(* CODESYS project ATV32_EIP_LMCx00C_V003.project
   Company: Schneider Electric
   DefaultNamespace: QuickMotionProgramming
   Title: QuickMotionProgramming
   Description: Demoproject for QuickMotionProgramming
   Author: Schneider Electric Automation GmbH
   Version: 1.0.6.0

Project tree, tasks and I/O mapping:
  LMC_PacDrive : PacDrive LMC 300/400/600C, Schneider Electric, order no. LMCx00C, version 1.51.10.0
    application Application
      libraries: PD_GlobalDiagnostics, 1.2.0.0 (Schneider Electric); PD_PacDriveLib, 1.4.9.0 (Schneider Electric); PD_AxisModule, 1.3.5.0 (Schneider Electric); PD_Template, 1.3.3.0 (Schneider Electric)
      task TASK_SR_MainMachine (cyclic, interval T#10ms, priority 8, watchdog T#100ms x 10) calls SR_MainMachine
      GlobalVariables/
        global variables RestoreAxisPosition
        global variables GlobalVariables_Machine
        global variables Global_ATV32
        global variables Logging
        global variables HardwareInOuts
        global variables InputVariablesSLB
        global variables InputVariablesExt
        global variables ExceptionHandling
        global variables Diagnostics
      ProjectDiagnostics/
        function FC_EtDiagExtUserToString [ST]
        data type ET_DiagExtUser
        data type ET_DiagExt
        function FC_EtDiagExtToString [ST]
      000 Program/
        00 Task Calls/
          program SR_MainMachine [LD]: Logic_ATV32
      Data Types/
        data type ET_Cmd
        data type ET_ATV32CmdWord
        data type ET_ATV32StatusWord
      300 EIP Utilities/
        function FC_EIPWriteWORDtoBYTES [ST]
        function FC_EIPReadWORDfromBYTES [ST]
    EPAS Mechatronic
    EPAS SERCOSIII Device Commissioning
    Message Logger
    SERCOSIII : SERCOS III Interface, Schneider Electric, version 1.51.10.0
      DRV_Master : Lexium LXM62 Drive, Schneider Electric, order no. LXM62DU60, LXM62DD15, LXM62DD27, LXM62DD45, LXM62DC13, version 1.51.10.0
          settings: ConfiguredPowerSupply = 'PSM_Lexium62'
      DRV_Axis1 : Lexium LXM62 Drive, Schneider Electric, order no. LXM62DU60, LXM62DD15, LXM62DD27, LXM62DD45, LXM62DC13, version 1.51.10.0
          settings: ConfiguredPowerSupply = 'PSM_Lexium62'
      DRV_Axis2 : Lexium LXM62 Drive, Schneider Electric, order no. LXM62DU60, LXM62DD15, LXM62DD27, LXM62DD45, LXM62DC13, version 1.51.10.0
          settings: ConfiguredPowerSupply = 'PSM_Lexium62'
      PSM_Lexium62 : Lexium LXM62 Power Supply, Schneider Electric, order no. LXM62PD84, LXM62PD20, version 1.51.10.0
    DIG_DigitalIn : Digital Inputs, Schneider Electric, version 1.51.10.0
      DI_11 : Input, Schneider Electric, version 1.51.10.0
      DI_2 : Input, Schneider Electric, version 1.51.10.0
      DI_10 : Input, Schneider Electric, version 1.51.10.0
      DI_19 : Input, Schneider Electric, version 1.51.10.0
      DI_5 : Input, Schneider Electric, version 1.51.10.0
      DI_17 : Input, Schneider Electric, version 1.51.10.0
      DI_0 : Input, Schneider Electric, version 1.51.10.0
      DI_8 : Input, Schneider Electric, version 1.51.10.0
      DI_1 : Input, Schneider Electric, version 1.51.10.0
      ADI_0 : Fast Input, Schneider Electric, version 1.51.10.0
      ADI_1 : Fast Input, Schneider Electric, version 1.51.10.0
      DI_9 : Input, Schneider Electric, version 1.51.10.0
      DI_12 : Input, Schneider Electric, version 1.51.10.0
      DI_15 : Input, Schneider Electric, version 1.51.10.0
      DI_6 : Input, Schneider Electric, version 1.51.10.0
      DI_13 : Input, Schneider Electric, version 1.51.10.0
      DI_14 : Input, Schneider Electric, version 1.51.10.0
      ADI_2 : Fast Input, Schneider Electric, version 1.51.10.0
      ADI_3 : Fast Input, Schneider Electric, version 1.51.10.0
      DI_7 : Input, Schneider Electric, version 1.51.10.0
      DI_4 : Input, Schneider Electric, version 1.51.10.0
      DI_16 : Input, Schneider Electric, version 1.51.10.0
      DI_18 : Input, Schneider Electric, version 1.51.10.0
      DI_3 : Input, Schneider Electric, version 1.51.10.0
    DQG_DigitalOut : Digital Outputs, Schneider Electric, version 1.51.10.0
        settings: DiagMask = 2#1111111100000000; OpenloadDiagMsk = 2#1111111100000000
      DQ_1 : Output, Schneider Electric, version 1.51.10.0
      DQ_0 : Output, Schneider Electric, version 1.51.10.0
      DQ_6 : Output, Schneider Electric, version 1.51.10.0
      DQ_4 : Output, Schneider Electric, version 1.51.10.0
      DQ_9 : Output, Schneider Electric, version 1.51.10.0
      DQ_13 : Output, Schneider Electric, version 1.51.10.0
      DQ_14 : Output, Schneider Electric, version 1.51.10.0
      DQ_15 : Output, Schneider Electric, version 1.51.10.0
      DQ_10 : Output, Schneider Electric, version 1.51.10.0
      DQ_5 : Output, Schneider Electric, version 1.51.10.0
      DQ_12 : Output, Schneider Electric, version 1.51.10.0
      DQ_11 : Output, Schneider Electric, version 1.51.10.0
      DQ_2 : Output, Schneider Electric, version 1.51.10.0
      DQ_3 : Output, Schneider Electric, version 1.51.10.0
      DQ_8 : Output, Schneider Electric, version 1.51.10.0
      DQ_7 : Output, Schneider Electric, version 1.51.10.0
    AI_0 : Analog Input, Schneider Electric, version 1.51.10.0
    AI_1 : Analog Input, Schneider Electric, version 1.51.10.0
    AQ_1 : Analog Output, Schneider Electric, version 1.51.10.0
    TPG_TPIn : Touch Probe Inputs, Schneider Electric, version 1.51.10.0
      TP_3 : Touch Probe Input, Schneider Electric, version 1.51.10.0
      TP_9 : Touch Probe Input, Schneider Electric, version 1.51.10.0
      TP_4 : Touch Probe Input, Schneider Electric, version 1.51.10.0
      TP_5 : Touch Probe Input, Schneider Electric, version 1.51.10.0
      TP_6 : Touch Probe Input, Schneider Electric, version 1.51.10.0
      TP_14 : Touch Probe Input, Schneider Electric, version 1.51.10.0
      TP_7 : Touch Probe Input, Schneider Electric, version 1.51.10.0
      TP_15 : Touch Probe Input, Schneider Electric, version 1.51.10.0
      TP_8 : Touch Probe Input, Schneider Electric, version 1.51.10.0
      TP_12 : Touch Probe Input, Schneider Electric, version 1.51.10.0
      TP_13 : Touch Probe Input, Schneider Electric, version 1.51.10.0
      TP_11 : Touch Probe Input, Schneider Electric, version 1.51.10.0
      TP_0 : Touch Probe Input, Schneider Electric, version 1.51.10.0
      TP_1 : Touch Probe Input, Schneider Electric, version 1.51.10.0
      TP_2 : Touch Probe Input, Schneider Electric, version 1.51.10.0
      TP_10 : Touch Probe Input, Schneider Electric, version 1.51.10.0
    AQ_0 : Analog Output, Schneider Electric, version 1.51.10.0
    LE_Master : Log. Encoder, Schneider Electric, version 1.51.10.0
    LE_Axis1 : Log. Encoder, Schneider Electric, version 1.51.10.0
    LE_Axis2 : Log. Encoder, Schneider Electric, version 1.51.10.0
    EIPS_Scanner : EtherNet-IP-Scanner, Schneider Electric, version 1.51.10.0
        settings: IPAddress = [16#C0,16#A8,16#01,16#0A]; SubnetMask = [16#FF,16#FF,16#FF,16#00]; GatewayAddress = [16#00,16#00,16#00,16#00]
      ATV32 : ATV32, Schneider Electric, version Major Revision=16#1, Minor Revision = 16#7
          settings: INITIALIZED = TRUE; IP address of Target = [16#C0,16#A8,16#01,16#14]; MAC address of Target = [16#00,16#00,16#00,16#00,16#00,16#00]; Keying.Check Minor Revision = FALSE; Number of Connections = 1; Connection Settings.Requested packet intervall (µs) = 10000; Connection Settings.OT Connection Parameters = 18450; Connection Settings.TO Connection Parameters = 10254; Connection Settings.Connection Flags = 1056; Connection Settings.Connection Path Size = 8; Connection Path = [16#20,16#04,16#24,16#05,16#2C,16#64,16#2C,16#65]
          input  Application.g_abATV32_1_StatusWordBytes[1] : BYTE  // Input0
          input  Application.g_abATV32_1_StatusWordBytes[2] : BYTE  // Input1
          input  Application.g_abATV32_1_ActVelocityBytes[1] : BYTE  // Input2
          input  Application.g_abATV32_1_ActVelocityBytes[2] : BYTE  // Input3
          output Application.g_abATV32_1_CommandWordBytes[1] : BYTE  // Output0
          output Application.g_abATV32_1_CommandWordBytes[2] : BYTE  // Output1
          output Application.g_abATV32_1_CmdVelocityBytes[1] : BYTE  // Output2
          output Application.g_abATV32_1_CmdVelocityBytes[2] : BYTE  // Output3
          unmapped channels: Input4, Input5, Input6, Input7, Input8, Input9, Input10, Input11, Output4, Output5, Output6, Output7, Output8, Output9, Output10, Output11
  Project Information/
    function GetVersion [ST]
    function GetBooleanProperty [ST]
    function GetTitle [ST]
    function GetVersionProperty [ST]
    function GetTextProperty [ST]
    function GetCompany [ST]
    function GetNumberProperty [ST]
  MainMachine
    DRV_Master
      Drive
    DRV_Axis2
      Drive
    DRV_Axis1
      Drive
    PSM_Lexium62
  MainMachine
    DRV_Master
      Drive
    DRV_Axis1
      Drive
    DRV_Axis2
      Drive
    PSM_Lexium62
  text list GlobalTextList
*)

// LMC_PacDrive/Application/ProjectDiagnostics/ET_DiagExtUser
{attribute 'qualified_only'}
TYPE ET_DiagExtUser :
(
(* Minimum value +0 *)
	Exception1FromEquipmentModule		:= 0,
	Exception2FromEquipmentModule		:= 1,
	
	Exception1FromMain					:= 2,
	Exception2FromMain					:= 3,
	Exception3FromMain					:= 4,
	Exception4FromMain					:= 5,
	Exception5FromMain					:= 6
)UDINT;
END_TYPE

// LMC_PacDrive/Application/ProjectDiagnostics/ET_DiagExt
{attribute 'qualified_only'}
TYPE ET_DiagExt :
(  
	(* Minimum value +0 *)
	Ok								:= 0,
	Disabled						:= 1,
	WaitUntilControllerFinishedBoot	:= 2,
	Initializing					:= 3,
	DeactivatingSubModules			:= 4,
	ExecuteStep						:= 5,
	WaitAtNegativeStep				:= 6,
	WaitCmdsDone					:= 7,
	WaitForCmd						:= 8,
	SubModuleInException			:= 9,
	ModuleControllerException		:= 10,
	UnknownStateModuleController	:= 11,
	
	SystemFatalException			:= 12,
	SystemException					:= 13,
	SystemWarning					:= 14,
	MainSystemEmergencyStop			:= 15,
	InvalidPointer					:= 16,	
	UpdateStructsException			:= 17,
	InitReactionsException			:= 18,
	InitSubModulesException			:= 19,
	DriveInvalid					:= 20,
	UnknownDiagExt					:= 21,
	
	Exception1FromVis				:= 22,
	Exception2FromVis				:= 23,
	Exception3FromVis				:= 24,
	Exception4FromVis				:= 25,
	Exception5FromVis				:= 26,
	
	DiagnosticsWarning					:= 27,
	WaitUntilDiagnosticsManagerReady	:= 28,
	WaitUntilDisabled					:= 29,
	WaitUntilDiagSourceRegistered		:= 30,
	WaitForCommunication				:= 31,
	DataSuccessfullyWritten				:= 32,
	WritingToFile						:= 33,
	FileIdInvalid						:= 34,
	CmdUnknown							:= 35,	
	UnexpectedFeedback					:= 36,
	UnknownDiagExtUser					:= 37,
	
	ExceptionListOverflow				:= 50
	
)UDINT;
END_TYPE

// LMC_PacDrive/Application/Data Types/ET_Cmd
{attribute 'qualified_only'}
TYPE ET_Cmd :
(	NoCmd				:= 0,

	(* TPL.Gc_udiUserCmdOffset : UDINT := 25000; // >= 25000: user defined Commands *)
	DriveEnableOn		:= 25999,
	DriveEnableOff		:= 25998,
	Init				:= 25997,
	Prepare				:= 25996,
	Production			:= 25995,
	Auto				:= 25994,
	BrakeRelease		:= 25993,
	Abort				:= 25992,
	Standby				:= 25991,
	Manual				:= 25990,
	Jogging				:= 25989,
	Hold				:= 25988,
	Stop				:= 25987,
	Start				:= 25986,
	HoldJM				:= 25985
);
END_TYPE

// LMC_PacDrive/Application/Data Types/ET_ATV32CmdWord
TYPE ET_ATV32CmdWord :
(
	Bit0_SwitchOn := 0,
	Bit1_EnableVoltage := 1,
	Bit2_QuickStop := 2,
	Bit3_EnableOperation := 3,
	Bit4_CmdUnused,
	Bit5_CmdUnused,
	Bit6_CmdUnused,
	Bit7_FaultReset,
	Bit8_Halt,
	Bit9_CmdUnused,
	Bit10_CmdUnused,
	Bit11_FwdRev,
	Bit12_CmdUnused,
	Bit13_CmdUnused,
	Bit14_CmdUnused,
	Bit15_CmdUnused
	
);
END_TYPE

// LMC_PacDrive/Application/Data Types/ET_ATV32StatusWord
TYPE ET_ATV32StatusWord :
(
	Bit0_ReadyToSwitchOn := 0,
	Bit1_SwitchedOn := 1,
	Bit2_OperationEnabled := 2,
	Bit3_Fault := 3,
	Bit4_VoltageEnabled,
	Bit5_QuickStop,
	Bit6_SwitchOnDisabled,
	Bit7_Warning,
	Bit8_StsUnused,
	Bit9_CmdViaNetwork,
	Bit10_TargetReached,
	Bit11_LimitActive,
	Bit12_StsUnused,
	Bit13_StsUnused,
	Bit14_StsUnused,
	Bit15_StsUnused
	
);
END_TYPE

// LMC_PacDrive/Application/GlobalVariables/RestoreAxisPosition
VAR_GLOBAL PERSISTENT RETAIN
	Grp_stRestorePositionMaster	: PDL.ST_AxisRestorePosition;
	Grp_stRestorePositionAxis1	: PDL.ST_AxisRestorePosition;
	Grp_stRestorePositionAxis2	: PDL.ST_AxisRestorePosition;
	Grp_stRestorePositionAxis3	: PDL.ST_AxisRestorePosition;
	Grp_stRestorePositionMaster2: PDL.ST_AxisRestorePosition;
	Grp_stRestorePositionAxis4	: PDL.ST_AxisRestorePosition;
	Grp_stRestorePositionAxis5	: PDL.ST_AxisRestorePosition;
	Grp_stRestorePositionAxis6	: PDL.ST_AxisRestorePosition;	
END_VAR

// LMC_PacDrive/Application/GlobalVariables/GlobalVariables_Machine
VAR_GLOBAL
	g_xAllServosHomeOk			:BOOL;
END_VAR

// LMC_PacDrive/Application/GlobalVariables/Global_ATV32
VAR_GLOBAL
	g_wATV32_1_CommandVelocity:		WORD;
	g_wATV32_1_ActVelocity:		WORD;

	g_abATV32_1_CommandWordBytes:	ARRAY[1..2] OF BYTE;
	g_axATV32_1CommandWord:			ARRAY[0..15] OF BOOL;
	g_wATV32_1_CommandWord:			WORD;

	g_abATV32_1_StatusWordBytes:	ARRAY[1..2] OF BYTE;
	g_axATV32_1StatusWord:			ARRAY[0..15] OF BOOL;
	g_wATV32_1_StatusWord:			WORD;
	
	g_abATV32_1_CmdVelocityBytes:	ARRAY[1..2] OF BYTE;
	g_abATV32_1_ActVelocityBytes:	ARRAY[1..2] OF BYTE;	
END_VAR

// LMC_PacDrive/Application/GlobalVariables/Logging
VAR_GLOBAL
	G_stLogDataList			: TPL.ST_LogDataList;			(* Global log data list *)
	G_stLogDataListAscii	: TPL.ST_LogDataListAscii;		(* Temp.list for save in XML format *)
	G_stLoggerInterface		: TPL.ST_LoggerInterface;		(* Interface between logger and main machine *)
END_VAR

// LMC_PacDrive/Application/GlobalVariables/HardwareInOuts
VAR_GLOBAL
	G_xMainsContactorOut 		(*-AT %QX0.0-*)	: BOOL;

	G_xEmergencyIn  			(*-AT %IX0.0-*)	: BOOL;
	G_xMainsContactorIn 		(*-AT %IX0.1-*)	: BOOL;
END_VAR

// LMC_PacDrive/Application/GlobalVariables/InputVariablesSLB
VAR_GLOBAL
	(* SoMachine Motion Logic Builder (SLB) input *)
	G_xStartSlb				 	: BOOL;
	G_xStopSlb					: BOOL;
	G_xPrepareSlb				: BOOL;
	G_xAutoSlb					: BOOL;
	G_xHoldSlb					: BOOL;
	G_xAbortSlb					: BOOL;
	G_xProductsOkSlb			: BOOL;
	G_xPowerOnSlb				: BOOL;
	G_xPowerOffSlb				: BOOL;
	G_xManualSlb				: BOOL;
	G_xJogMachineSlb			: BOOL;
	G_xDiagQuitSlb				: BOOL;
	G_xEmergencySlb				: BOOL := TRUE;
	G_xJogForwSlb				: BOOL;
	G_xJogBackSlb				: BOOL;
	G_xBrakeReleaseSlb			: BOOL;
	
	G_udiManualModuleSelect		: UDINT;

	G_xDoEnableVis				: BOOL;

	G_xDoPrepare 				: BOOL;
	G_xDoAuto	 				: BOOL;
	G_xDoManual 				: BOOL;
	G_xDoJogMachine 			: BOOL;
	G_xDoBrakeRelease			: BOOL;

	G_xPrepareActive 			: BOOL;
	G_xAutoActive	 			: BOOL;
	G_xManualActive 			: BOOL;
	G_xJogMachineActive 		: BOOL;
	G_xBrakeReleaseActive		: BOOL;
END_VAR

// LMC_PacDrive/Application/GlobalVariables/InputVariablesExt
VAR_GLOBAL
	(* Extern / HMI input *)
	G_xStartExt			: BOOL;
	G_xStopExt			: BOOL;
	G_xPrepareExt		: BOOL;
	G_xAutoExt			: BOOL;
	G_xHoldExt			: BOOL;
	G_xAbortExt			: BOOL;
	G_xProductsOkExt	: BOOL;
	G_xPowerOnExt		: BOOL;
	G_xPowerOffExt		: BOOL;
	G_xManualExt		: BOOL;
	G_xJogMachineExt	: BOOL;
	G_xDiagQuitExt		: BOOL;
	G_xJogForwExt		: BOOL;
	G_xJogBackExt		: BOOL;
	G_xBrakeReleaseExt	: BOOL;
END_VAR

// LMC_PacDrive/Application/GlobalVariables/ExceptionHandling
VAR_GLOBAL
	G_stExceptionList		: TPL.ST_ExceptionList;
END_VAR

// LMC_PacDrive/Application/GlobalVariables/Diagnostics
VAR_GLOBAL
	G_stDiagnosticsToApplicationMarkerarea AT %MB0 : TPL.ST_DiagnosticsToApplicationMarkerArea;
END_VAR

// LMC_PacDrive/Application/000 Program/00 Task Calls/SR_MainMachine
PROGRAM SR_MainMachine
VAR
END_VAR

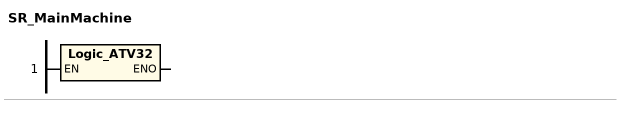
// NETWORK 1
Logic_ATV32();

ACTION Logic_ATV32:




g_wATV32_1_CommandWord := PDL.FC_PackWord(
											i_xB15:= g_axATV32_1CommandWord[Bit15_CmdUnused], 
											i_xB14:= g_axATV32_1CommandWord[Bit14_CmdUnused], 
											i_xB13:= g_axATV32_1CommandWord[Bit13_CmdUnused], 
											i_xB12:= g_axATV32_1CommandWord[Bit12_CmdUnused], 
											i_xB11:= g_axATV32_1CommandWord[Bit11_FwdRev], 
											i_xB10:= g_axATV32_1CommandWord[Bit10_CmdUnused], 
											i_xB09:= g_axATV32_1CommandWord[Bit9_CmdUnused], 
											i_xB08:= g_axATV32_1CommandWord[Bit8_Halt], 
											i_xB07:= g_axATV32_1CommandWord[Bit7_FaultReset], 
											i_xB06:= g_axATV32_1CommandWord[Bit6_CmdUnused], 
											i_xB05:= g_axATV32_1CommandWord[Bit5_CmdUnused], 
											i_xB04:= g_axATV32_1CommandWord[Bit4_CmdUnused], 
											i_xB03:= g_axATV32_1CommandWord[Bit3_EnableOperation], 
											i_xB02:= g_axATV32_1CommandWord[Bit2_QuickStop], 
											i_xB01:= g_axATV32_1CommandWord[Bit1_EnableVoltage], 
											i_xB00:= g_axATV32_1CommandWord[Bit0_SwitchOn]);

								
// Write the Command Word - FC_EIPWriteWORDtoBYTES allows us to send a word vlaue to two consecutive bytes in memory
FC_EIPWriteWORDtoBYTES(pdiSourceWord:= ADR(g_wATV32_1_CommandWord), pDestByte:=ADR(g_abATV32_1_CommandWordBytes[1]) );											

// Write the Command Velocity - FC_EIPWriteWORDtoBYTES allows us to send a word vlaue to two consecutive bytes in memory
FC_EIPWriteWORDtoBYTES(pdiSourceWord:= ADR(g_wATV32_1_CommandVelocity), pDestByte:=ADR(g_abATV32_1_CmdVelocityBytes[1]) );

// Read The Status Word - FC_EIPReadWORDFromBYTES allows us to read a word vlaue to two consecutive bytes in memory
g_wATV32_1_StatusWord := FC_EIPReadWORDfromBYTES(pByteSource:=ADR(g_abATV32_1_StatusWordBytes[1]));
	
PDL.FC_UnpackWord(i_wInput:= g_wATV32_1_StatusWord, 
				  	q_xB15=> g_axATV32_1StatusWord[Bit15_StsUnused], 
				  	q_xB14=> g_axATV32_1StatusWord[Bit14_StsUnused], 
					q_xB13=> g_axATV32_1StatusWord[Bit13_StsUnused], 
					q_xB12=> g_axATV32_1StatusWord[Bit12_StsUnused], 
					q_xB11=> g_axATV32_1StatusWord[Bit11_LimitActive], 
					q_xB10=> g_axATV32_1StatusWord[Bit10_TargetReached], 
					q_xB09=> g_axATV32_1StatusWord[Bit9_CmdViaNetwork], 
					q_xB08=> g_axATV32_1StatusWord[Bit8_StsUnused], 
					q_xB07=> g_axATV32_1StatusWord[Bit7_Warning], 
					q_xB06=> g_axATV32_1StatusWord[Bit6_SwitchOnDisabled], 
					q_xB05=> g_axATV32_1StatusWord[Bit5_QuickStop], 
					q_xB04=> g_axATV32_1StatusWord[Bit4_VoltageEnabled], 
					q_xB03=> g_axATV32_1StatusWord[Bit3_Fault], 
					q_xB02=> g_axATV32_1StatusWord[Bit2_OperationEnabled], 
					q_xB01=> g_axATV32_1StatusWord[Bit1_SwitchedOn], 
					q_xB00=> g_axATV32_1StatusWord[Bit0_ReadyToSwitchOn]);
					
// Read Actual Velocity - FC_EIPReadWORDFromBYTES allows us to read a word vlaue to two consecutive bytes in memory					
					
g_wATV32_1_ActVelocity := FC_EIPReadWORDfromBYTES(pByteSource:=ADR(g_abATV32_1_ActVelocityBytes[1]));
END_ACTION

END_PROGRAM

// LMC_PacDrive/Application/300 EIP Utilities/FC_EIPWriteWORDtoBYTES
FUNCTION FC_EIPWriteWORDtoBYTES : WORD
(* This function will write to a WORD to 2 succesive Bytes starting from the input var "pdiDestByte"
	When calling the function, "pDestByte" should be the address of an index from an ARRAY OF BYTE, then the function
	will build the WORD based on the data from the index you start with plus the next indexes in order from the array.

	Example:

	Declaration:    MyByteArray:			ARRAY[1..128] OF BYTE;

	Function Call:        FC_EIPWriteWORDtoBYTES(pdiSourceWord:= ADR(MyWORDVariable), pDestByte:= ADR(MyByteArray[1]));
*)
VAR_INPUT
	pdiSourceWord:		POINTER TO WORD;
	pDestByte:			POINTER TO WORD;
END_VAR
VAR
END_VAR

pDestByte^ := pdiSourceWord^;

END_FUNCTION

// LMC_PacDrive/Application/300 EIP Utilities/FC_EIPReadWORDfromBYTES
FUNCTION FC_EIPReadWORDfromBYTES : WORD
(* 

	Exp:
	Declaration:    MyByteArray:			ARRAY[1..128] OF BYTE;

	Function Call:        OutputDINTVaraible := FC_EIPReadWORDfromBYTES(ADR(MyByteArray[1]);
*)
VAR_INPUT
	pByteSource:		POINTER TO WORD;
END_VAR
VAR
END_VAR

FC_EIPReadWORDfromBYTES := pByteSource^;

END_FUNCTION

// Project Information/GetVersion
// This function has been automatically generated from the project information.
{attribute 'signature_flag' := '1073741824'}
{attribute 'register_in_runtime'}
FUNCTION GetVersion : VERSION
VAR_INPUT
	
END_VAR

GetVersion.uiMajor := 1;
GetVersion.uiMinor := 0;
GetVersion.uiServicePack := 6;
GetVersion.uiPatch := 0;

END_FUNCTION

// Project Information/GetBooleanProperty
// This function has been automatically generated from the project information.
{attribute 'signature_flag' := '1073741824'}
{attribute 'register_in_runtime'}
FUNCTION GetBooleanProperty : BOOL
VAR_INPUT
	stKey: WSTRING;
END_VAR

GetBooleanProperty := FALSE;

END_FUNCTION

// Project Information/GetTitle
// This function has been automatically generated from the project information.
{attribute 'signature_flag' := '1073741824'}
{attribute 'register_in_runtime'}
FUNCTION GetTitle : WSTRING
VAR_INPUT
	
END_VAR

GetTitle := "QuickMotionProgramming";

END_FUNCTION

// Project Information/GetVersionProperty
// This function has been automatically generated from the project information.
{attribute 'signature_flag' := '1073741824'}
{attribute 'register_in_runtime'}
FUNCTION GetVersionProperty : VERSION
VAR_INPUT
	stKey: WSTRING;
END_VAR

IF stKey = "Version" THEN
	GetVersionProperty.uiMajor := 1;
	GetVersionProperty.uiMinor := 0;
	GetVersionProperty.uiServicePack := 6;
	GetVersionProperty.uiPatch := 0;
ELSE
	GetVersionProperty.uiMajor := 0;
	GetVersionProperty.uiMinor := 0;
	GetVersionProperty.uiServicePack := 0;
	GetVersionProperty.uiPatch := 0;
END_IF

END_FUNCTION

// Project Information/GetTextProperty
// This function has been automatically generated from the project information.
{attribute 'signature_flag' := '1073741824'}
{attribute 'register_in_runtime'}
FUNCTION GetTextProperty : WSTRING
VAR_INPUT
	stKey: WSTRING;
END_VAR

IF stKey = "Author" THEN
	GetTextProperty := "Schneider Electric Automation GmbH";
ELSIF stKey = "Company" THEN
	GetTextProperty := "Schneider Electric";
ELSIF stKey = "DefaultNamespace" THEN
	GetTextProperty := "QuickMotionProgramming";
ELSIF stKey = "Description" THEN
	GetTextProperty := "Demoproject for QuickMotionProgramming";
ELSIF stKey = "Project" THEN
	GetTextProperty := "ATV32_EIP_LMCx00C_V003";
ELSIF stKey = "Title" THEN
	GetTextProperty := "QuickMotionProgramming";
ELSE
	GetTextProperty := "";
END_IF

END_FUNCTION

// Project Information/GetCompany
// This function has been automatically generated from the project information.
{attribute 'signature_flag' := '1073741824'}
{attribute 'register_in_runtime'}
FUNCTION GetCompany : WSTRING
VAR_INPUT
	
END_VAR

GetCompany := "Schneider Electric";

END_FUNCTION

// Project Information/GetNumberProperty
// This function has been automatically generated from the project information.
{attribute 'signature_flag' := '1073741824'}
{attribute 'register_in_runtime'}
FUNCTION GetNumberProperty : DINT
VAR_INPUT
	stKey: WSTRING;
END_VAR

GetNumberProperty := 0;

END_FUNCTION

// LMC_PacDrive/Application/ProjectDiagnostics/FC_EtDiagExtUserToString
FUNCTION FC_EtDiagExtUserToString : STRING[80]

VAR_INPUT
	i_etDiagExt : ET_DiagExtUser;
END_VAR

VAR_OUTPUT
	q_etDiag	: GD.ET_Diag := GD.ET_Diag.Ok;
	q_etDiagExt	: ET_DiagExt := ET_DiagExt.Ok;
END_VAR

VAR
END_VAR

CASE i_etDiagExt OF
	ET_DiagExtUser.Exception1FromEquipmentModule	: FC_EtDiagExtUserToString := 'Exception1FromEquipmentModule';
	ET_DiagExtUser.Exception2FromEquipmentModule	: FC_EtDiagExtUserToString := 'Exception2FromEquipmentModule';
	
	ET_DiagExtUser.Exception1FromMain				: FC_EtDiagExtUserToString := 'Exception1FromMain';
	ET_DiagExtUser.Exception2FromMain				: FC_EtDiagExtUserToString := 'Exception2FromMain';
	ET_DiagExtUser.Exception3FromMain				: FC_EtDiagExtUserToString := 'Exception3FromMain';
	ET_DiagExtUser.Exception4FromMain				: FC_EtDiagExtUserToString := 'Exception4FromMain';
	ET_DiagExtUser.Exception5FromMain				: FC_EtDiagExtUserToString := 'Exception5FromMain';
ELSE
	FC_EtDiagExtUserToString := CONCAT('Unkown ET_DiagExtUser ', UDINT_TO_STRING(i_etDiagExt));
		
	q_etDiag	:= GD.ET_Diag.InputParameterInvalid;
	q_etDiagExt	:= ET_DiagExt.UnknownDiagExtUser;
END_CASE

END_FUNCTION

// LMC_PacDrive/Application/ProjectDiagnostics/FC_EtDiagExtToString
FUNCTION FC_EtDiagExtToString : STRING[80]

VAR_INPUT
	i_etDiagExt : ET_DiagExt;
END_VAR

VAR_OUTPUT
	q_etDiag	: GD.ET_Diag := GD.ET_Diag.Ok;
	q_etDiagExt	: ET_DiagExt := ET_DiagExt.Ok;
END_VAR

VAR
END_VAR

CASE i_etDiagExt OF
	ET_DiagExt.Ok:								FC_EtDiagExtToString := 'Ok';
	ET_DiagExt.Disabled:						FC_EtDiagExtToString := 'Disabled';
	ET_DiagExt.WaitUntilControllerFinishedBoot:	FC_EtDiagExtToString := 'WaitUntilControllerFinishedBoot';
	ET_DiagExt.Initializing:					FC_EtDiagExtToString := 'Initializing';
	ET_DiagExt.DeactivatingSubModules:			FC_EtDiagExtToString := 'DeactivatingSubModules';
	ET_DiagExt.ExecuteStep:						FC_EtDiagExtToString := 'ExecuteStep';
	ET_DiagExt.WaitAtNegativeStep:				FC_EtDiagExtToString := 'WaitAtNegativeStep';
	ET_DiagExt.WaitCmdsDone:					FC_EtDiagExtToString := 'WaitCmdsDone';
	ET_DiagExt.WaitForCmd:						FC_EtDiagExtToString := 'WaitForCmd';
	ET_DiagExt.SubModuleInException:			FC_EtDiagExtToString := 'SubModuleInException';
	ET_DiagExt.ModuleControllerException:		FC_EtDiagExtToString := 'ModuleControllerException';
	ET_DiagExt.UnknownStateModuleController:	FC_EtDiagExtToString := 'UnknownStateModuleController';
	
	ET_DiagExt.SystemFatalException:			FC_EtDiagExtToString := 'SystemFatalException';
	ET_DiagExt.SystemException:					FC_EtDiagExtToString := 'SystemException';
	ET_DiagExt.SystemWarning:					FC_EtDiagExtToString := 'SystemWarning';
	ET_DiagExt.MainSystemEmergencyStop:			FC_EtDiagExtToString := 'MainSystemEmergencyStop';
	ET_DiagExt.InvalidPointer:					FC_EtDiagExtToString := 'InvalidPointer';
	ET_DiagExt.UpdateStructsException:			FC_EtDiagExtToString := 'UpdateStructsException';
	ET_DiagExt.InitReactionsException:			FC_EtDiagExtToString := 'InitReactionsException';
	ET_DiagExt.InitSubModulesException:			FC_EtDiagExtToString := 'InitSubModulesException';
	ET_DiagExt.DriveInvalid:					FC_EtDiagExtToString := 'DriveInvalid';
	ET_DiagExt.UnknownDiagExt:					FC_EtDiagExtToString := 'UnknownDiagExt';

	ET_DiagExt.Exception1FromVis:				FC_EtDiagExtToString := 'Exception1FromVis';
	ET_DiagExt.Exception2FromVis:				FC_EtDiagExtToString := 'Exception2FromVis';
	ET_DiagExt.Exception3FromVis:				FC_EtDiagExtToString := 'Exception3FromVis';
	ET_DiagExt.Exception4FromVis:				FC_EtDiagExtToString := 'Exception4FromVis';
	ET_DiagExt.Exception5FromVis:				FC_EtDiagExtToString := 'Exception5FromVis';
	
	ET_DiagExt.DiagnosticsWarning:				FC_EtDiagExtToString := 'DiagnosticsWarning';
	ET_DiagExt.WaitUntilDiagnosticsManagerReady:FC_EtDiagExtToString := 'WaitUntilDiagnosticsManagerReady';
	ET_DiagExt.WaitUntilDisabled:				FC_EtDiagExtToString := 'WaitUntilDisabled';
	ET_DiagExt.WaitUntilDiagSourceRegistered:	FC_EtDiagExtToString := 'WaitUntilDiagSourceRegistered';
	ET_DiagExt.WaitForCommunication:			FC_EtDiagExtToString := 'WaitForCommunication';
	ET_DiagExt.DataSuccessfullyWritten:			FC_EtDiagExtToString := 'DataSuccessfullyWritten';
	ET_DiagExt.WritingToFile:					FC_EtDiagExtToString := 'WritingToFile';
	ET_DiagExt.FileIdInvalid:					FC_EtDiagExtToString := 'FileIdInvalid';
	ET_DiagExt.CmdUnknown:						FC_EtDiagExtToString := 'CmdUnknown';
	ET_DiagExt.UnexpectedFeedback:				FC_EtDiagExtToString := 'UnexpectedFeedback';
	ET_DiagExt.UnknownDiagExtUser:				FC_EtDiagExtToString := 'UnknownDiagExtUser';
	
	ET_DiagExt.ExceptionListOverflow:			FC_EtDiagExtToString := 'ExceptionListOverflow';
ELSE
	FC_EtDiagExtToString := CONCAT('Unkown ET_DiagExt ', UDINT_TO_STRING(i_etDiagExt));
		
	q_etDiag	:= GD.ET_Diag.InputParameterInvalid;
	q_etDiagExt	:= ET_DiagExt.UnknownDiagExt;
END_CASE

END_FUNCTION
